{attribute 'GeneratedUsingTerminal: EL5152-0000-0016'}
{attribute addProperty BoxType "EL5152-0000-0016"}
{attribute addProperty Id "Set_counterAT %Q*BOOL1Set_counter_valueAT %Q*UINT2"}
{attribute addProperty CRC "610056523"}
{attribute addProperty Size "3"}
TYPE ENC_Control_compact_Channel_245CB94B EXTENDS OutputBase_10CEE7DE :
STRUCT
	{attribute addProperty Name "Set_counter"}
	Set_counter AT %Q* : BOOL;
	{attribute addProperty Name "Set_counter_value"}
	Set_counter_value AT %Q* : UINT;
END_STRUCT
END_TYPE

(* stored: Version 1.2.0.0, ProductVersion 3.1.4024.9
   DUT ENC_Control_compact_Channel_245CB94B: Id {dbb6620a-d34d-4992-a09f-765cb5a23ae8} *)
